{attribute 'qualified_only'}
{attribute 'strict'}
TYPE nCompresorTypes :
(
	_8P0		:= 0,
	Volvo_CMA	:= 1
);
END_TYPE

(* stored: Version 1.1.0.1, ProductVersion 3.1.4024.12
   DUT nCompresorTypes: Id {48ee39d1-910e-47ef-96f1-619f8b881951} *)
